// TwinCAT 3 PLC project GJA_TDF
// ProgramVersion: 3.1.4022.7
// libraries:
//   Tc2_MC2, * (Beckhoff Automation GmbH)
//   Tc2_MC2_FlyingSaw, * (Beckhoff Automation GmbH)
//   Tc2_Standard, * (Beckhoff Automation GmbH)
//   Tc2_System, * (Beckhoff Automation GmbH)
//   Tc3_Module, * (Beckhoff Automation GmbH)
// project tree:
//   GVLs/ GVL1001_CommonSignal.TcGVL, GVL20_NC.TcGVL, Param_NC.TcGVL
//   / PlcTask.TcTTO
//   POUs/100 NC/ P01_AxesControl.TcPOU
//   POUs/ MAIN.TcPOU
// real-time tasks:
//   TASK PlcTask: cycle T#10ms, priority 20, ADS port 350
// motion (NC):
//   TASK NC-Task 1 SAF: cycle T#2ms, priority 4, ADS port 501
//   TASK NC-Task 1 SVB: cycle T#10ms, priority 8, ADS port 511
//   AXIS Axis 1 (id 1)
//     OtherSettings: AllowMotionCmdToSlave=true
//     encoder EncType=1
//     drive DrvType=5
//       Analog: ScaleFactorActTorque=0.1
//     controller CtrType=1
//       CtrPara: PriorControlFactor=1
//         Observer: BandWidth=20
//   AXIS Axis 2 (id 2)
//     OtherSettings: AllowMotionCmdToSlave=true
//     encoder EncType=1
//     drive DrvType=5
//       Analog: ScaleFactorActTorque=0.1
//     controller CtrType=1
//       CtrPara: PriorControlFactor=1
//         Observer: BandWidth=20
//   AXIS Axis 3 (id 3)
//     OtherSettings: AllowMotionCmdToSlave=true
//     encoder EncType=1
//     drive DrvType=5
//       Analog: ScaleFactorActTorque=0.1
//     controller CtrType=1
//       CtrPara: PriorControlFactor=1
//         Observer: BandWidth=20
//   AXIS Axis 4 (id 4)
//     OtherSettings: AllowMotionCmdToSlave=true
//     encoder EncType=1
//     drive DrvType=5
//       Analog: ScaleFactorActTorque=0.1
//     controller CtrType=1
//       CtrPara: PriorControlFactor=1
//         Observer: BandWidth=20

CONFIGURATION GJA_TDF
    RESOURCE PLC ON TwinCAT3
        TASK PlcTask(INTERVAL := T#10ms, PRIORITY := 20);
        PROGRAM MAIN WITH PlcTask : MAIN;
    END_RESOURCE
END_CONFIGURATION

// ---- GVLs/GVL1001_CommonSignal.TcGVL
{attribute 'qualified_only'}
VAR_GLOBAL
	gxPowerOn		:BOOL; 	//系统上电
	gxPowerOff		:BOOL;	//系统断电
	grOverride		:REAL;	//override
	
	gxEnable		:BOOL;	//使能信号
	gbSysReady		:BOOL;	//系统准备就绪
	gbAlarm			:BOOL;	//系统故障
	
	
END_VAR

// ---- GVLs/GVL20_NC.TcGVL
{attribute 'qualified_only'}
VAR_GLOBAL
	gastAxis	:ARRAY[1..Param_NC.gc_NC_Max] OF AXIS_REF;
END_VAR

// ---- GVLs/Param_NC.TcGVL
{attribute 'qualified_only'}
VAR_GLOBAL CONSTANT
	gc_NC_Max	:INT	:=4;
END_VAR

// ---- POUs/MAIN.TcPOU
PROGRAM MAIN
VAR
	bInit	:BOOL;
END_VAR

P01_AxesControl();

END_PROGRAM

// ---- POUs/100 NC/P01_AxesControl.TcPOU
PROGRAM P01_AxesControl
VAR
	// 系统上电
	fbMC_Power		:ARRAY[1.. Param_NC.gc_NC_Max] OF MC_Power;
	i				: INT	:= 1;
END_VAR

FOR i:=1 TO Param_NC.gc_NC_Max DO
fbMC_Power[i](
	Axis:= GVL20_NC.gastAxis[i], 
	Enable:= GVL1001_CommonSignal.gxEnable AND GVL1001_CommonSignal.gxPowerOn, 
	Enable_Positive:= TRUE, 
	Enable_Negative:= TRUE, 
	Override:= GVL1001_CommonSignal.grOverride, 
	BufferMode:= , 
	Options:= , 
	Status=> , 
	Busy=> , 
	Active=> , 
	Error=> , 
	ErrorID=> );
END_FOR

END_PROGRAM
